Copyright (c) 2019 Manuel Goester, Michael Witt, Klaus Kammerer
Institute of Databases and Information Systems, Ulm University, Germany

Permission is hereby granted, free of charge, to any person obtaining a copy 
of this software and associated documentation files (the "Software"), to deal 
in the Software without restriction, including without limitation the rights 
to use, copy, modify, merge, publish, distribute, sublicense, and/or sell 
copies of the Software, and to permit persons to whom the Software is 
furnished to do so, subject to the following conditions:

The above copyright notice and this permission notice shall be included in 
all copies or substantial portions of the Software.

THE SOFTWARE IS PROVIDED "AS IS", WITHOUT WARRANTY OF ANY KIND, EXPRESS OR 
IMPLIED, INCLUDING BUT NOT LIMITED TO THE WARRANTIES OF MERCHANTABILITY, 
FITNESS FOR A PARTICULAR PURPOSE AND NONINFRINGEMENT. IN NO EVENT SHALL THE 
AUTHORS OR COPYRIGHT HOLDERS BE LIABLE FOR ANY CLAIM, DAMAGES OR OTHER 
LIABILITY, WHETHER IN AN ACTION OF CONTRACT, TORT OR OTHERWISE, ARISING FROM, 
OUT OF OR IN CONNECTION WITH THE SOFTWARE OR THE USE OR OTHER DEALINGS 
IN THE SOFTWARE.
*)
FUNCTION_BLOCK HR_TAKE_W_FROM_CONVEYOR
VAR_INPUT
	w: Workpiece;
END_VAR
VAR_OUTPUT
END_VAR
VAR
	step: INT := 1;
	hr_move: HR_MOVE;
	fin: BOOL := FALSE;
	stepFin: BOOL := FALSE;
END_VAR

fin := FALSE;
CASE step OF
	1:	// forward if not already there
		IF NOT(HR.sCFront) THEN
			HR.mCForward := TRUE;
		ELSE
			HR.mCForward := FALSE;
			step := step + 1;
		END_IF
	2:	// backwards
		IF HR.lbIn THEN
			HR.mCbBackward := TRUE;
		ELSE
			HR.mCbBackward := FALSE;
			step := step + 1; 
		END_IF
	3:	// up
		hr_move(x := 0, y := -26);
		stepFin := hr_move.fin;
		IF stepFin THEN
			step := step + 1;
			stepFin := FALSE;
		END_IF
	4:	// back
		IF NOT(HR.sCBack) THEN
			HR.mCBackward := TRUE;
		ELSE
			HR.mCBackward := FALSE;
			step := step + 1;
		END_IF
	5:	// finished
		fin := TRUE;
		step := 1;
		stepFin := FALSE;
END_CASE

END_FUNCTION_BLOCK

// Device/Application/HR/FBs/HR_PUT_W
(*
	HR puts down a workpiece into rack or at conveyor
	
Copyright (c) 2019 Manuel Goester, Michael Witt, Klaus Kammerer
Institute of Databases and Information Systems, Ulm University, Germany

Permission is hereby granted, free of charge, to any person obtaining a copy 
of this software and associated documentation files (the "Software"), to deal 
in the Software without restriction, including without limitation the rights 
to use, copy, modify, merge, publish, distribute, sublicense, and/or sell 
copies of the Software, and to permit persons to whom the Software is 
furnished to do so, subject to the following conditions:

The above copyright notice and this permission notice shall be included in 
all copies or substantial portions of the Software.

THE SOFTWARE IS PROVIDED "AS IS", WITHOUT WARRANTY OF ANY KIND, EXPRESS OR 
IMPLIED, INCLUDING BUT NOT LIMITED TO THE WARRANTIES OF MERCHANTABILITY, 
FITNESS FOR A PARTICULAR PURPOSE AND NONINFRINGEMENT. IN NO EVENT SHALL THE 
AUTHORS OR COPYRIGHT HOLDERS BE LIABLE FOR ANY CLAIM, DAMAGES OR OTHER 
LIABILITY, WHETHER IN AN ACTION OF CONTRACT, TORT OR OTHERWISE, ARISING FROM, 
OUT OF OR IN CONNECTION WITH THE SOFTWARE OR THE USE OR OTHER DEALINGS 
IN THE SOFTWARE.
*)
FUNCTION_BLOCK HR_PUT_W
VAR_INPUT
END_VAR
VAR_OUTPUT
END_VAR
VAR
	step: INT := 1;
	hr_move: HR_MOVE;
	fin: BOOL := FALSE;
	stepFin: BOOL := FALSE;
END_VAR

CASE step OF
	1:	// forward
		fin := FALSE;
		IF NOT(HR.sCFront) THEN
			HR.mCForward := TRUE;
		ELSE
			HR.mCForward := FALSE;
			step := step + 1;
		END_IF
	2:	// down
		hr_move(x := 0 , y := 16);
		stepFin := hr_move.fin;
		IF stepFin THEN
			step := step + 1;
			stepFin := FALSE;
		END_IF
	3:	// back
		IF NOT(HR.sCBack) THEN
			HR.mCBackward := TRUE;
		ELSE
			HR.mCBackward := FALSE;
			step := step + 1;
		END_IF
	4:	// finished
		fin := TRUE;
		step := 1;
END_CASE

END_FUNCTION_BLOCK

// Device/Application/HR/HR_MULTI_MODE
PROGRAM HR_MULTI_MODE
VAR
	fin: BOOL;
	hr_get: HR_GET_W;
	hr_store: HR_STORE_W;
	hr_put_w_on_conveyor: HR_PUT_W_ON_CONVEYOR;
	
	// for GET_W
	// calibrate y axis of rack every 3th workpiece
	calibrateYAxis: INT := 0;
	calibarteYAxisCounted: BOOL := FALSE;
	step: INT := 1;
	timer: TON;
END_VAR

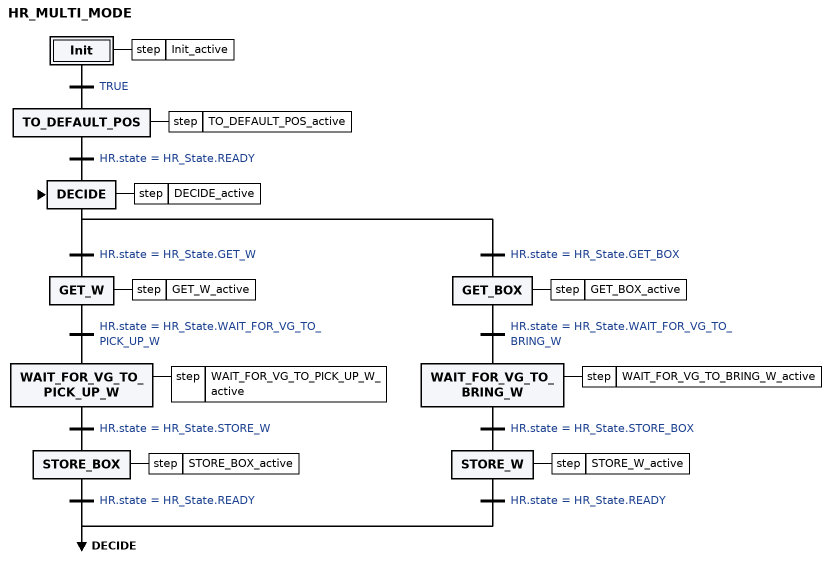
INITIAL_STEP Init:
    Init_active(N);  // step action
END_STEP
TRANSITION FROM Init TO TO_DEFAULT_POS
    := TRUE;
END_TRANSITION
STEP TO_DEFAULT_POS:
    TO_DEFAULT_POS_active(N);  // step action
END_STEP
TRANSITION FROM TO_DEFAULT_POS TO DECIDE
    := HR.state = HR_State.READY;
END_TRANSITION
STEP DECIDE:
    DECIDE_active(N);  // step action
END_STEP
TRANSITION FROM DECIDE TO GET_W
    := HR.state = HR_State.GET_W;
END_TRANSITION
STEP GET_W:
    GET_W_active(N);  // step action
END_STEP
TRANSITION FROM GET_W TO WAIT_FOR_VG_TO_PICK_UP_W
    := HR.state = HR_State.WAIT_FOR_VG_TO_PICK_UP_W;
END_TRANSITION
STEP WAIT_FOR_VG_TO_PICK_UP_W:
    WAIT_FOR_VG_TO_PICK_UP_W_active(N);  // step action
END_STEP
TRANSITION FROM WAIT_FOR_VG_TO_PICK_UP_W TO STORE_BOX
    := HR.state = HR_State.STORE_W;
END_TRANSITION
STEP STORE_BOX:
    STORE_BOX_active(N);  // step action
END_STEP
TRANSITION FROM STORE_BOX TO DECIDE
    := HR.state = HR_State.READY;
END_TRANSITION
TRANSITION FROM DECIDE TO GET_BOX
    := HR.state = HR_State.GET_BOX;
END_TRANSITION
STEP GET_BOX:
    GET_BOX_active(N);  // step action
END_STEP
TRANSITION FROM GET_BOX TO WAIT_FOR_VG_TO_BRING_W
    := HR.state = HR_State.WAIT_FOR_VG_TO_BRING_W;
END_TRANSITION
STEP WAIT_FOR_VG_TO_BRING_W:
    WAIT_FOR_VG_TO_BRING_W_active(N);  // step action
END_STEP
TRANSITION FROM WAIT_FOR_VG_TO_BRING_W TO STORE_W
    := HR.state = HR_State.STORE_BOX;
END_TRANSITION
STEP STORE_W:
    STORE_W_active(N);  // step action
END_STEP
TRANSITION FROM STORE_W TO DECIDE
    := HR.state = HR_State.READY;
END_TRANSITION

ACTION STORE_BOX_active:
(*
Copyright (c) 2019 Manuel Goester, Michael Witt, Klaus Kammerer
Institute of Databases and Information Systems, Ulm University, Germany

Permission is hereby granted, free of charge, to any person obtaining a copy 
of this software and associated documentation files (the "Software"), to deal 
in the Software without restriction, including without limitation the rights 
to use, copy, modify, merge, publish, distribute, sublicense, and/or sell 
copies of the Software, and to permit persons to whom the Software is 
furnished to do so, subject to the following conditions:

The above copyright notice and this permission notice shall be included in 
all copies or substantial portions of the Software.

THE SOFTWARE IS PROVIDED "AS IS", WITHOUT WARRANTY OF ANY KIND, EXPRESS OR 
IMPLIED, INCLUDING BUT NOT LIMITED TO THE WARRANTIES OF MERCHANTABILITY, 
FITNESS FOR A PARTICULAR PURPOSE AND NONINFRINGEMENT. IN NO EVENT SHALL THE 
AUTHORS OR COPYRIGHT HOLDERS BE LIABLE FOR ANY CLAIM, DAMAGES OR OTHER 
LIABILITY, WHETHER IN AN ACTION OF CONTRACT, TORT OR OTHERWISE, ARISING FROM, 
OUT OF OR IN CONNECTION WITH THE SOFTWARE OR THE USE OR OTHER DEALINGS 
IN THE SOFTWARE.
*)
IF NOT fin THEN
	// store box in rack
	hr_store(w := HR.currW);
	fin := hr_store.fin;
ELSE
	fin := FALSE;
	HR.state := HR_State.READY;
END_IF
END_ACTION

ACTION GET_W_active:
(*
Copyright (c) 2019 Manuel Goester, Michael Witt, Klaus Kammerer
Institute of Databases and Information Systems, Ulm University, Germany

Permission is hereby granted, free of charge, to any person obtaining a copy 
of this software and associated documentation files (the "Software"), to deal 
in the Software without restriction, including without limitation the rights 
to use, copy, modify, merge, publish, distribute, sublicense, and/or sell 
copies of the Software, and to permit persons to whom the Software is 
furnished to do so, subject to the following conditions:

The above copyright notice and this permission notice shall be included in 
all copies or substantial portions of the Software.

THE SOFTWARE IS PROVIDED "AS IS", WITHOUT WARRANTY OF ANY KIND, EXPRESS OR 
IMPLIED, INCLUDING BUT NOT LIMITED TO THE WARRANTIES OF MERCHANTABILITY, 
FITNESS FOR A PARTICULAR PURPOSE AND NONINFRINGEMENT. IN NO EVENT SHALL THE 
AUTHORS OR COPYRIGHT HOLDERS BE LIABLE FOR ANY CLAIM, DAMAGES OR OTHER 
LIABILITY, WHETHER IN AN ACTION OF CONTRACT, TORT OR OTHERWISE, ARISING FROM, 
OUT OF OR IN CONNECTION WITH THE SOFTWARE OR THE USE OR OTHER DEALINGS 
IN THE SOFTWARE.
*)
// increment y calibration counter
IF NOT(calibarteYAxisCounted) THEN
	calibrateYAxis := calibrateYAxis + 1;
	calibarteYAxisCounted := TRUE;
END_IF

IF calibrateYAxis >= 3 THEN
	// calibrate y axis
	IF NOT(HR.sVertical) THEN
		HR.mVerticalUp := TRUE;
	ELSE
		Hr.mVerticalUp := FALSE;
		Hr.cY := 0;
		calibrateYAxis := 0;
	END_IF
ELSE
	CASE step OF
		1:
			// get w from rack
			IF NOT fin THEN
				hr_get(w:= HR.currW);
				fin := hr_get.fin;
			ELSE
				fin := FALSE;
				step := step + 1;
			END_IF
		2:
			// put w on conveyor
			hr_put_w_on_conveyor(w := HR.currW);
			fin := hr_put_w_on_conveyor.fin;	
			IF fin THEN
				step := step + 1;
				fin := FALSE;
			END_IF
		3:
			// bring it to VG in conveyor
			IF HR.lbOut THEN
				HR.mCbForward := TRUE;
			ELSE
				// start 1 sec timer to drive conveyor 1 sec longer to be sure that box is at outside pos
				timer(IN:= TRUE, PT := T#1S);
				IF NOT(timer.Q = FALSE AND timer.IN) THEN
					timer(IN:= FALSE);
					HR.mCbForward := FALSE;
					step := step + 1; 
				END_IF
			END_IF
		4:
			// finished
			step := 1;
			HR.state := HR_State.WAIT_FOR_VG_TO_PICK_UP_W;
			calibarteYAxisCounted := FALSE;
			// bend VG pointers to current workpiece of HR
			VG.bIdx := TC.currBatchJobIdx;
			VG.wIdx := TC.batchJobQueue.batchJobs[TC.currBatchJobIdx].nextNotProcessedIdx;
			VG.currW := TC.batchJobQueue.batchJobs[VG.bIdx].workpieces[VG.wIdx];
	END_CASE
END_IF
END_ACTION

ACTION WAIT_FOR_VG_TO_PICK_UP_W_active:
(*
Copyright (c) 2019 Manuel Goester, Michael Witt, Klaus Kammerer
Institute of Databases and Information Systems, Ulm University, Germany

Permission is hereby granted, free of charge, to any person obtaining a copy 
of this software and associated documentation files (the "Software"), to deal 
in the Software without restriction, including without limitation the rights 
to use, copy, modify, merge, publish, distribute, sublicense, and/or sell 
copies of the Software, and to permit persons to whom the Software is 
furnished to do so, subject to the following conditions:

The above copyright notice and this permission notice shall be included in 
all copies or substantial portions of the Software.

THE SOFTWARE IS PROVIDED "AS IS", WITHOUT WARRANTY OF ANY KIND, EXPRESS OR 
IMPLIED, INCLUDING BUT NOT LIMITED TO THE WARRANTIES OF MERCHANTABILITY, 
FITNESS FOR A PARTICULAR PURPOSE AND NONINFRINGEMENT. IN NO EVENT SHALL THE 
AUTHORS OR COPYRIGHT HOLDERS BE LIABLE FOR ANY CLAIM, DAMAGES OR OTHER 
LIABILITY, WHETHER IN AN ACTION OF CONTRACT, TORT OR OTHERWISE, ARISING FROM, 
OUT OF OR IN CONNECTION WITH THE SOFTWARE OR THE USE OR OTHER DEALINGS 
IN THE SOFTWARE.
*)
IF VG.state = VG_State.TO_FUR_PUT_W OR VG.state = VG_State.TO_EJECT THEN
	HR.state := HR_State.STORE_W;
	HR.decidedToTakeANewW := FALSE;
END_IF
END_ACTION

ACTION GET_BOX_active:
(*
Copyright (c) 2019 Manuel Goester, Michael Witt, Klaus Kammerer
Institute of Databases and Information Systems, Ulm University, Germany

Permission is hereby granted, free of charge, to any person obtaining a copy 
of this software and associated documentation files (the "Software"), to deal 
in the Software without restriction, including without limitation the rights 
to use, copy, modify, merge, publish, distribute, sublicense, and/or sell 
copies of the Software, and to permit persons to whom the Software is 
furnished to do so, subject to the following conditions:

The above copyright notice and this permission notice shall be included in 
all copies or substantial portions of the Software.

THE SOFTWARE IS PROVIDED "AS IS", WITHOUT WARRANTY OF ANY KIND, EXPRESS OR 
IMPLIED, INCLUDING BUT NOT LIMITED TO THE WARRANTIES OF MERCHANTABILITY, 
FITNESS FOR A PARTICULAR PURPOSE AND NONINFRINGEMENT. IN NO EVENT SHALL THE 
AUTHORS OR COPYRIGHT HOLDERS BE LIABLE FOR ANY CLAIM, DAMAGES OR OTHER 
LIABILITY, WHETHER IN AN ACTION OF CONTRACT, TORT OR OTHERWISE, ARISING FROM, 
OUT OF OR IN CONNECTION WITH THE SOFTWARE OR THE USE OR OTHER DEALINGS 
IN THE SOFTWARE.
*)
CASE step OF
	1:
		IF NOT fin THEN
			hr_get(w:= HR.currW);
			fin := hr_get.fin;
		ELSE
			step := step + 1;
			fin := FALSE;
		END_IF
	2:
		// put w on conveyor
		hr_put_w_on_conveyor(w := HR.currW);
		fin := hr_put_w_on_conveyor.fin;	
		IF fin THEN
			step := step + 1;
			fin := FALSE;
		END_IF
	3:
		// bring it to VG in conveyor
		IF HR.lbOut THEN
			HR.mCbForward := TRUE;
		ELSE
			// start 1 sec timer to drive conveyor 1 sec longer to be sure that box is at outside pos
			timer(IN:= TRUE, PT := T#1S);
			IF NOT(timer.Q = FALSE AND timer.IN) THEN
				timer(IN:= FALSE);
				HR.mCbForward := FALSE;
				step := step + 1; 
			END_IF
		END_IF
	4:
		// finished
		step := 1;
		HR.state := HR_State.WAIT_FOR_VG_TO_BRING_W;
END_CASE
END_ACTION

ACTION DECIDE_active:
(*
Copyright (c) 2019 Manuel Goester, Michael Witt, Klaus Kammerer
Institute of Databases and Information Systems, Ulm University, Germany

Permission is hereby granted, free of charge, to any person obtaining a copy 
of this software and associated documentation files (the "Software"), to deal 
in the Software without restriction, including without limitation the rights 
to use, copy, modify, merge, publish, distribute, sublicense, and/or sell 
copies of the Software, and to permit persons to whom the Software is 
furnished to do so, subject to the following conditions:

The above copyright notice and this permission notice shall be included in 
all copies or substantial portions of the Software.

THE SOFTWARE IS PROVIDED "AS IS", WITHOUT WARRANTY OF ANY KIND, EXPRESS OR 
IMPLIED, INCLUDING BUT NOT LIMITED TO THE WARRANTIES OF MERCHANTABILITY, 
FITNESS FOR A PARTICULAR PURPOSE AND NONINFRINGEMENT. IN NO EVENT SHALL THE 
AUTHORS OR COPYRIGHT HOLDERS BE LIABLE FOR ANY CLAIM, DAMAGES OR OTHER 
LIABILITY, WHETHER IN AN ACTION OF CONTRACT, TORT OR OTHERWISE, ARISING FROM, 
OUT OF OR IN CONNECTION WITH THE SOFTWARE OR THE USE OR OTHER DEALINGS 
IN THE SOFTWARE.
*)

// if sl positions free or if not free if workpiece will not be ejected 
// AND VG is not storing
// AND HR does not already decided to take a new workpiece
// THEN 
IF ((SL.lbRed AND SL.lbWhite AND SL.lbBlue) OR (SL.currW.format.ejectEnabled AND NOT(SL.currW.state = W_State.NULL))) AND NOT(VG.storeW) AND NOT(decidedToTakeANewW) THEN
	HR.bIdx := 0;
	HR.wIdx := 0;
	HR.currW := TC.nullW;
	HR.decidedToTakeANewW := TRUE;
	VG.storeW := FALSE;
ELSIF HR.decidedToTakeANewW THEN
	// get new w out of rack
	IF TC.state = TC_state.W_LOADED THEN
		// set pointers to make sure that they are set
		Hr.bIdx := TC.currBatchJobIdx;
		Hr.wIdx := TC.batchJobQueue.batchJobs[TC.currBatchJobIdx].nextNotProcessedIdx;
		HR.currW := TC.batchJobQueue.batchJobs[Hr.bIdx].workpieces[Hr.wIdx];
		// workpiece is loaded, start production
		HR.state := HR_State.GET_W;
		// signalise that production starts
		TC.state := TC_State.WAIT_UNTIL_W_FINISHED;
	ELSE
		// no workpiece loaded, load it now
		TC.state := TC_State.LOAD_NEXT_W;
	END_IF
ELSE
	// prevent misconduct when a workpiece is still lying in one of the three spots at SL, although the application got reset
	IF NOT(VG.bIdx = 0) THEN
		// get empty box out of rack
		// set workpiece to get the right box from rack
		IF NOT(SL.lbWhite) OR NOT(SL.lbRed) OR NOT(SL.lbBlue) THEN
			HR.bIdx := SL.bIdx;
			HR.wIdx := SL.wIdx;
			HR.currW := SL.currW;
		ELSE
			HR.bIdx := VG.bIdx;
			HR.wIdx := VG.wIdx;
			HR.currW := VG.currW;
		END_IF
		HR.state := HR_State.GET_BOX;
		// reset flag
		VG.storeW := FALSE;
		END_IF
END_IF
END_ACTION

ACTION STORE_W_active:
(*
Copyright (c) 2019 Manuel Goester, Michael Witt, Klaus Kammerer
Institute of Databases and Information Systems, Ulm University, Germany

Permission is hereby granted, free of charge, to any person obtaining a copy 
of this software and associated documentation files (the "Software"), to deal 
in the Software without restriction, including without limitation the rights 
to use, copy, modify, merge, publish, distribute, sublicense, and/or sell 
copies of the Software, and to permit persons to whom the Software is 
furnished to do so, subject to the following conditions:

The above copyright notice and this permission notice shall be included in 
all copies or substantial portions of the Software.

THE SOFTWARE IS PROVIDED "AS IS", WITHOUT WARRANTY OF ANY KIND, EXPRESS OR 
IMPLIED, INCLUDING BUT NOT LIMITED TO THE WARRANTIES OF MERCHANTABILITY, 
FITNESS FOR A PARTICULAR PURPOSE AND NONINFRINGEMENT. IN NO EVENT SHALL THE 
AUTHORS OR COPYRIGHT HOLDERS BE LIABLE FOR ANY CLAIM, DAMAGES OR OTHER 
LIABILITY, WHETHER IN AN ACTION OF CONTRACT, TORT OR OTHERWISE, ARISING FROM, 
OUT OF OR IN CONNECTION WITH THE SOFTWARE OR THE USE OR OTHER DEALINGS 
IN THE SOFTWARE.
*)
IF NOT fin THEN
	// store workpiece in rack
	hr_store(w := HR.currW);
	fin := hr_store.fin;
ELSE
	fin := FALSE;
	HR.state := HR_State.READY;
END_IF
END_ACTION

ACTION WAIT_FOR_VG_TO_BRING_W_active:
(*
Copyright (c) 2019 Manuel Goester, Michael Witt, Klaus Kammerer
Institute of Databases and Information Systems, Ulm University, Germany

Permission is hereby granted, free of charge, to any person obtaining a copy 
of this software and associated documentation files (the "Software"), to deal 
in the Software without restriction, including without limitation the rights 
to use, copy, modify, merge, publish, distribute, sublicense, and/or sell 
copies of the Software, and to permit persons to whom the Software is 
furnished to do so, subject to the following conditions:

The above copyright notice and this permission notice shall be included in 
all copies or substantial portions of the Software.

THE SOFTWARE IS PROVIDED "AS IS", WITHOUT WARRANTY OF ANY KIND, EXPRESS OR 
IMPLIED, INCLUDING BUT NOT LIMITED TO THE WARRANTIES OF MERCHANTABILITY, 
FITNESS FOR A PARTICULAR PURPOSE AND NONINFRINGEMENT. IN NO EVENT SHALL THE 
AUTHORS OR COPYRIGHT HOLDERS BE LIABLE FOR ANY CLAIM, DAMAGES OR OTHER 
LIABILITY, WHETHER IN AN ACTION OF CONTRACT, TORT OR OTHERWISE, ARISING FROM, 
OUT OF OR IN CONNECTION WITH THE SOFTWARE OR THE USE OR OTHER DEALINGS 
IN THE SOFTWARE.
*)
IF VG.state = VG_State.TO_HR_PUT_W_FINISHED OR HR.currW.format.ejectEnabled THEN
	HR.state := HR_State.STORE_BOX;
END_IF
END_ACTION

ACTION Init_active:
(*
Copyright (c) 2019 Manuel Goester, Michael Witt, Klaus Kammerer
Institute of Databases and Information Systems, Ulm University, Germany

Permission is hereby granted, free of charge, to any person obtaining a copy 
of this software and associated documentation files (the "Software"), to deal 
in the Software without restriction, including without limitation the rights 
to use, copy, modify, merge, publish, distribute, sublicense, and/or sell 
copies of the Software, and to permit persons to whom the Software is 
furnished to do so, subject to the following conditions:

The above copyright notice and this permission notice shall be included in 
all copies or substantial portions of the Software.

THE SOFTWARE IS PROVIDED "AS IS", WITHOUT WARRANTY OF ANY KIND, EXPRESS OR 
IMPLIED, INCLUDING BUT NOT LIMITED TO THE WARRANTIES OF MERCHANTABILITY, 
FITNESS FOR A PARTICULAR PURPOSE AND NONINFRINGEMENT. IN NO EVENT SHALL THE 
AUTHORS OR COPYRIGHT HOLDERS BE LIABLE FOR ANY CLAIM, DAMAGES OR OTHER 
LIABILITY, WHETHER IN AN ACTION OF CONTRACT, TORT OR OTHERWISE, ARISING FROM, 
OUT OF OR IN CONNECTION WITH THE SOFTWARE OR THE USE OR OTHER DEALINGS 
IN THE SOFTWARE.
*)
calibrateYAxis := 0;
calibarteYAxisCounted := FALSE;
END_ACTION

ACTION TO_DEFAULT_POS_active:
(*
Copyright (c) 2019 Manuel Goester, Michael Witt, Klaus Kammerer
Institute of Databases and Information Systems, Ulm University, Germany

Permission is hereby granted, free of charge, to any person obtaining a copy 
of this software and associated documentation files (the "Software"), to deal 
in the Software without restriction, including without limitation the rights 
to use, copy, modify, merge, publish, distribute, sublicense, and/or sell 
copies of the Software, and to permit persons to whom the Software is 
furnished to do so, subject to the following conditions:

The above copyright notice and this permission notice shall be included in 
all copies or substantial portions of the Software.

THE SOFTWARE IS PROVIDED "AS IS", WITHOUT WARRANTY OF ANY KIND, EXPRESS OR 
IMPLIED, INCLUDING BUT NOT LIMITED TO THE WARRANTIES OF MERCHANTABILITY, 
FITNESS FOR A PARTICULAR PURPOSE AND NONINFRINGEMENT. IN NO EVENT SHALL THE 
AUTHORS OR COPYRIGHT HOLDERS BE LIABLE FOR ANY CLAIM, DAMAGES OR OTHER 
LIABILITY, WHETHER IN AN ACTION OF CONTRACT, TORT OR OTHERWISE, ARISING FROM, 
OUT OF OR IN CONNECTION WITH THE SOFTWARE OR THE USE OR OTHER DEALINGS 
IN THE SOFTWARE.
*)
// returns High Rack TOWER to its default start position
// set "ausleger" arm to default position
IF HR.sCBack = FALSE THEN
	HR.mCBackward := TRUE;
ELSE 
	HR.mCBackward := FALSE;
	// set tower vertical position to max UP as well as horizontal position max RIGHT
	IF HR.sHorizontal = FALSE THEN
		HR.mHorizontalRight := TRUE;
	ELSE
		HR.mHorizontalRight := FALSE;
	END_IF
	
	IF HR.sVertical = FALSE THEN
		HR.mVerticalUp := TRUE;
	ELSE
		HR.mVerticalUp := FALSE;
	END_IF
END_IF

IF HR.sHorizontal AND HR.sVertical AND HR.sCBack THEN
	HR.cX := 0;
	HR.cY := 0;
	HR.state := HR_State.READY;
END_IF
END_ACTION

END_PROGRAM

// Device/Application/HR/HR_SORTING_MODE
PROGRAM HR_SORTING_MODE
VAR
	hr_switch_ws: HR_SWITCH_WS;
	fin: BOOL;
END_VAR

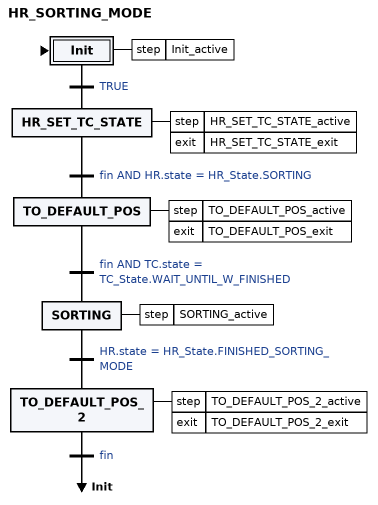
INITIAL_STEP Init:
    Init_active(N);  // step action
END_STEP
TRANSITION FROM Init TO HR_SET_TC_STATE
    := TRUE;
END_TRANSITION
STEP HR_SET_TC_STATE:
    HR_SET_TC_STATE_active(N);  // step action
    HR_SET_TC_STATE_exit(P0);  // exit action
END_STEP
TRANSITION FROM HR_SET_TC_STATE TO TO_DEFAULT_POS
    := fin AND HR.state = HR_State.SORTING;
END_TRANSITION
STEP TO_DEFAULT_POS:
    TO_DEFAULT_POS_active(N);  // step action
    TO_DEFAULT_POS_exit(P0);  // exit action
END_STEP
TRANSITION FROM TO_DEFAULT_POS TO SORTING
    := fin AND TC.state = TC_State.WAIT_UNTIL_W_FINISHED;
END_TRANSITION
STEP SORTING:
    SORTING_active(N);  // step action
END_STEP
TRANSITION FROM SORTING TO TO_DEFAULT_POS_2
    := HR.state = HR_State.FINISHED_SORTING_MODE;
END_TRANSITION
STEP TO_DEFAULT_POS_2:
    TO_DEFAULT_POS_2_active(N);  // step action
    TO_DEFAULT_POS_2_exit(P0);  // exit action
END_STEP
TRANSITION FROM TO_DEFAULT_POS_2 TO Init
    := fin;
END_TRANSITION

ACTION SORTING_active:
(*
Copyright (c) 2019 Manuel Goester, Michael Witt, Klaus Kammerer
Institute of Databases and Information Systems, Ulm University, Germany

Permission is hereby granted, free of charge, to any person obtaining a copy 
of this software and associated documentation files (the "Software"), to deal 
in the Software without restriction, including without limitation the rights 
to use, copy, modify, merge, publish, distribute, sublicense, and/or sell 
copies of the Software, and to permit persons to whom the Software is 
furnished to do so, subject to the following conditions:

The above copyright notice and this permission notice shall be included in 
all copies or substantial portions of the Software.

THE SOFTWARE IS PROVIDED "AS IS", WITHOUT WARRANTY OF ANY KIND, EXPRESS OR 
IMPLIED, INCLUDING BUT NOT LIMITED TO THE WARRANTIES OF MERCHANTABILITY, 
FITNESS FOR A PARTICULAR PURPOSE AND NONINFRINGEMENT. IN NO EVENT SHALL THE 
AUTHORS OR COPYRIGHT HOLDERS BE LIABLE FOR ANY CLAIM, DAMAGES OR OTHER 
LIABILITY, WHETHER IN AN ACTION OF CONTRACT, TORT OR OTHERWISE, ARISING FROM, 
OUT OF OR IN CONNECTION WITH THE SOFTWARE OR THE USE OR OTHER DEALINGS 
IN THE SOFTWARE.
*)
IF NOT(fin) THEN
	hr_switch_ws(w1 := TC.batchJobQueue.batchJobs[TC.currBatchJobIdx].workpieces[TC.batchJobQueue.batchJobs[TC.currBatchJobIdx].nextNotProcessedIdx], w2 := TC.batchJobQueue.batchJobs[TC.currBatchJobIdx].workpieces[TC.batchJobQueue.batchJobs[TC.currBatchJobIdx].nextNotProcessedIdx+1]);
	fin := hr_switch_ws.fin;
ELSE
	// sorting finished
	fin := FALSE;
	HR.state := HR_State.FINISHED_SORTING_MODE;
END_IF
END_ACTION

ACTION TO_DEFAULT_POS_exit:
(*
Copyright (c) 2019 Manuel Goester, Michael Witt, Klaus Kammerer
Institute of Databases and Information Systems, Ulm University, Germany

Permission is hereby granted, free of charge, to any person obtaining a copy 
of this software and associated documentation files (the "Software"), to deal 
in the Software without restriction, including without limitation the rights 
to use, copy, modify, merge, publish, distribute, sublicense, and/or sell 
copies of the Software, and to permit persons to whom the Software is 
furnished to do so, subject to the following conditions:

The above copyright notice and this permission notice shall be included in 
all copies or substantial portions of the Software.

THE SOFTWARE IS PROVIDED "AS IS", WITHOUT WARRANTY OF ANY KIND, EXPRESS OR 
IMPLIED, INCLUDING BUT NOT LIMITED TO THE WARRANTIES OF MERCHANTABILITY, 
FITNESS FOR A PARTICULAR PURPOSE AND NONINFRINGEMENT. IN NO EVENT SHALL THE 
AUTHORS OR COPYRIGHT HOLDERS BE LIABLE FOR ANY CLAIM, DAMAGES OR OTHER 
LIABILITY, WHETHER IN AN ACTION OF CONTRACT, TORT OR OTHERWISE, ARISING FROM, 
OUT OF OR IN CONNECTION WITH THE SOFTWARE OR THE USE OR OTHER DEALINGS 
IN THE SOFTWARE.
*)
fin := FALSE;
END_ACTION

ACTION TO_DEFAULT_POS_active:
(*
Copyright (c) 2019 Manuel Goester, Michael Witt, Klaus Kammerer
Institute of Databases and Information Systems, Ulm University, Germany

Permission is hereby granted, free of charge, to any person obtaining a copy 
of this software and associated documentation files (the "Software"), to deal 
in the Software without restriction, including without limitation the rights 
to use, copy, modify, merge, publish, distribute, sublicense, and/or sell 
copies of the Software, and to permit persons to whom the Software is 
furnished to do so, subject to the following conditions:

The above copyright notice and this permission notice shall be included in 
all copies or substantial portions of the Software.

THE SOFTWARE IS PROVIDED "AS IS", WITHOUT WARRANTY OF ANY KIND, EXPRESS OR 
IMPLIED, INCLUDING BUT NOT LIMITED TO THE WARRANTIES OF MERCHANTABILITY, 
FITNESS FOR A PARTICULAR PURPOSE AND NONINFRINGEMENT. IN NO EVENT SHALL THE 
AUTHORS OR COPYRIGHT HOLDERS BE LIABLE FOR ANY CLAIM, DAMAGES OR OTHER 
LIABILITY, WHETHER IN AN ACTION OF CONTRACT, TORT OR OTHERWISE, ARISING FROM, 
OUT OF OR IN CONNECTION WITH THE SOFTWARE OR THE USE OR OTHER DEALINGS 
IN THE SOFTWARE.
*)
// get HR to its default position
IF HR.sCBack = FALSE THEN
	HR.mCBackward := TRUE;
ELSE 
	HR.mCBackward := FALSE;
	// set tower vertical position to max UP as well as horizontal position max RIGHT
	IF HR.sHorizontal = FALSE THEN
		HR.mHorizontalRight := TRUE;
	ELSE
		HR.mHorizontalRight := FALSE;
		HR.cX := 0;
	END_IF
	
	IF HR.sVertical = FALSE THEN
		HR.mVerticalUp := TRUE;
	ELSE
		HR.mVerticalUp := FALSE;
		HR.cY := 0;
	END_IF
END_IF

IF HR.sHorizontal AND HR.sVertical AND HR.sCBack THEN
	// finished
	fin := TRUE;
END_IF
END_ACTION

ACTION Init_active:

END_ACTION

ACTION HR_SET_TC_STATE_active:
(*
Copyright (c) 2019 Manuel Goester, Michael Witt, Klaus Kammerer
Institute of Databases and Information Systems, Ulm University, Germany

Permission is hereby granted, free of charge, to any person obtaining a copy 
of this software and associated documentation files (the "Software"), to deal 
in the Software without restriction, including without limitation the rights 
to use, copy, modify, merge, publish, distribute, sublicense, and/or sell 
copies of the Software, and to permit persons to whom the Software is 
furnished to do so, subject to the following conditions:

The above copyright notice and this permission notice shall be included in 
all copies or substantial portions of the Software.

THE SOFTWARE IS PROVIDED "AS IS", WITHOUT WARRANTY OF ANY KIND, EXPRESS OR 
IMPLIED, INCLUDING BUT NOT LIMITED TO THE WARRANTIES OF MERCHANTABILITY, 
FITNESS FOR A PARTICULAR PURPOSE AND NONINFRINGEMENT. IN NO EVENT SHALL THE 
AUTHORS OR COPYRIGHT HOLDERS BE LIABLE FOR ANY CLAIM, DAMAGES OR OTHER 
LIABILITY, WHETHER IN AN ACTION OF CONTRACT, TORT OR OTHERWISE, ARISING FROM, 
OUT OF OR IN CONNECTION WITH THE SOFTWARE OR THE USE OR OTHER DEALINGS 
IN THE SOFTWARE.
*)
IF NOT(fin) THEN
	IF TC.state = TC_State.W_LOADED THEN
		TC.state := TC_State.WAIT_UNTIL_W_FINISHED;
		fin := TRUE;
	ELSE
		// load a new workpiece
		TC.state := TC_State.LOAD_NEXT_W;
	END_IF
END_IF
END_ACTION

ACTION HR_SET_TC_STATE_exit:
(*
Copyright (c) 2019 Manuel Goester, Michael Witt, Klaus Kammerer
Institute of Databases and Information Systems, Ulm University, Germany

Permission is hereby granted, free of charge, to any person obtaining a copy 
of this software and associated documentation files (the "Software"), to deal 
in the Software without restriction, including without limitation the rights 
to use, copy, modify, merge, publish, distribute, sublicense, and/or sell 
copies of the Software, and to permit persons to whom the Software is 
furnished to do so, subject to the following conditions:

The above copyright notice and this permission notice shall be included in 
all copies or substantial portions of the Software.

THE SOFTWARE IS PROVIDED "AS IS", WITHOUT WARRANTY OF ANY KIND, EXPRESS OR 
IMPLIED, INCLUDING BUT NOT LIMITED TO THE WARRANTIES OF MERCHANTABILITY, 
FITNESS FOR A PARTICULAR PURPOSE AND NONINFRINGEMENT. IN NO EVENT SHALL THE 
AUTHORS OR COPYRIGHT HOLDERS BE LIABLE FOR ANY CLAIM, DAMAGES OR OTHER 
LIABILITY, WHETHER IN AN ACTION OF CONTRACT, TORT OR OTHERWISE, ARISING FROM, 
OUT OF OR IN CONNECTION WITH THE SOFTWARE OR THE USE OR OTHER DEALINGS 
IN THE SOFTWARE.
*)
fin := FALSE;
END_ACTION

ACTION TO_DEFAULT_POS_2_exit:
(*
Copyright (c) 2019 Manuel Goester, Michael Witt, Klaus Kammerer
Institute of Databases and Information Systems, Ulm University, Germany

Permission is hereby granted, free of charge, to any person obtaining a copy 
of this software and associated documentation files (the "Software"), to deal 
in the Software without restriction, including without limitation the rights 
to use, copy, modify, merge, publish, distribute, sublicense, and/or sell 
copies of the Software, and to permit persons to whom the Software is 
furnished to do so, subject to the following conditions:

The above copyright notice and this permission notice shall be included in 
all copies or substantial portions of the Software.

THE SOFTWARE IS PROVIDED "AS IS", WITHOUT WARRANTY OF ANY KIND, EXPRESS OR 
IMPLIED, INCLUDING BUT NOT LIMITED TO THE WARRANTIES OF MERCHANTABILITY, 
FITNESS FOR A PARTICULAR PURPOSE AND NONINFRINGEMENT. IN NO EVENT SHALL THE 
AUTHORS OR COPYRIGHT HOLDERS BE LIABLE FOR ANY CLAIM, DAMAGES OR OTHER 
LIABILITY, WHETHER IN AN ACTION OF CONTRACT, TORT OR OTHERWISE, ARISING FROM, 
OUT OF OR IN CONNECTION WITH THE SOFTWARE OR THE USE OR OTHER DEALINGS 
IN THE SOFTWARE.
*)
fin := FALSE;
END_ACTION

ACTION TO_DEFAULT_POS_2_active:
(*
Copyright (c) 2019 Manuel Goester, Michael Witt, Klaus Kammerer
Institute of Databases and Information Systems, Ulm University, Germany

Permission is hereby granted, free of charge, to any person obtaining a copy 
of this software and associated documentation files (the "Software"), to deal 
in the Software without restriction, including without limitation the rights 
to use, copy, modify, merge, publish, distribute, sublicense, and/or sell 
copies of the Software, and to permit persons to whom the Software is 
furnished to do so, subject to the following conditions:

The above copyright notice and this permission notice shall be included in 
all copies or substantial portions of the Software.

THE SOFTWARE IS PROVIDED "AS IS", WITHOUT WARRANTY OF ANY KIND, EXPRESS OR 
IMPLIED, INCLUDING BUT NOT LIMITED TO THE WARRANTIES OF MERCHANTABILITY, 
FITNESS FOR A PARTICULAR PURPOSE AND NONINFRINGEMENT. IN NO EVENT SHALL THE 
AUTHORS OR COPYRIGHT HOLDERS BE LIABLE FOR ANY CLAIM, DAMAGES OR OTHER 
LIABILITY, WHETHER IN AN ACTION OF CONTRACT, TORT OR OTHERWISE, ARISING FROM, 
OUT OF OR IN CONNECTION WITH THE SOFTWARE OR THE USE OR OTHER DEALINGS 
IN THE SOFTWARE.
*)
// get HR to its default position
// needed, if a job multi / single mode batch job will be executed after ths batch
IF HR.sCBack = FALSE THEN
	HR.mCBackward := TRUE;
ELSE 
	HR.mCBackward := FALSE;
	// set tower vertical position to max UP as well as horizontal position max RIGHT
	IF HR.sHorizontal = FALSE THEN
		HR.mHorizontalRight := TRUE;
	ELSE
		HR.mHorizontalRight := FALSE;
		HR.cX := 0;
	END_IF
	
	IF HR.sVertical = FALSE THEN
		HR.mVerticalUp := TRUE;
	ELSE
		HR.mVerticalUp := FALSE;
		HR.cY := 0;
	END_IF
END_IF

IF HR.sHorizontal AND HR.sVertical AND HR.sCBack THEN
	// finished
	fin := TRUE;
END_IF
END_ACTION

END_PROGRAM

// Device/Application/HR/FBs/HR_SWITCH_WS
(*
	This Function Block gets two workpieces as input and switches their positions in the rack
	
Copyright (c) 2019 Manuel Goester, Michael Witt, Klaus Kammerer
Institute of Databases and Information Systems, Ulm University, Germany

Permission is hereby granted, free of charge, to any person obtaining a copy 
of this software and associated documentation files (the "Software"), to deal 
in the Software without restriction, including without limitation the rights 
to use, copy, modify, merge, publish, distribute, sublicense, and/or sell 
copies of the Software, and to permit persons to whom the Software is 
furnished to do so, subject to the following conditions:

The above copyright notice and this permission notice shall be included in 
all copies or substantial portions of the Software.

THE SOFTWARE IS PROVIDED "AS IS", WITHOUT WARRANTY OF ANY KIND, EXPRESS OR 
IMPLIED, INCLUDING BUT NOT LIMITED TO THE WARRANTIES OF MERCHANTABILITY, 
FITNESS FOR A PARTICULAR PURPOSE AND NONINFRINGEMENT. IN NO EVENT SHALL THE 
AUTHORS OR COPYRIGHT HOLDERS BE LIABLE FOR ANY CLAIM, DAMAGES OR OTHER 
LIABILITY, WHETHER IN AN ACTION OF CONTRACT, TORT OR OTHERWISE, ARISING FROM, 
OUT OF OR IN CONNECTION WITH THE SOFTWARE OR THE USE OR OTHER DEALINGS 
IN THE SOFTWARE.
*)
FUNCTION_BLOCK HR_SWITCH_WS
VAR_INPUT
	// first workpiece
	w1: Workpiece;
	// second workpiece
	w2: Workpiece;
END_VAR
VAR_OUTPUT
END_VAR
VAR
	stepFin : BOOL;
	step: INT := 1;
	hr_move_to_pos: HR_MOVE_TO_POS;
	hr_get_w: HR_GET_W;
	hr_take_w: HR_TAKE_W;
	hr_put_w: HR_PUT_W;
	fin: BOOL;
END_VAR

fin := FALSE;
CASE step OF
	1:	// get w1 out of rack and bring it to conveyor
		IF NOT(stepFin) THEN
			hr_get_w(w := w1);
			stepFin := hr_get_w.fin;
		ELSE
			stepFin := FALSE;
			step := step + 1;
		END_IF
	2:	// put down w1 at conveyor
		IF NOT(stepFin) THEN
			hr_put_w();
			stepFin := hr_put_w.fin;
		ELSE
			stepFin := FALSE;
			step := step + 1;
		END_IF
	3:	// move to w2 position in rack
		IF NOT(stepFin) THEN
			hr_move_to_pos(pos := w2.startPos, upOrDown := RackPos.DOWN);	
			stepFin := hr_move_to_pos.fin;
		ELSE
			stepFin := FALSE;
			step := step + 1;
		END_IF
	4:	// pick up w2
		IF NOT(stepFin) THEN
			hr_take_w();
			stepFin := hr_take_w.fin;
		ELSE
			stepFin := FALSE;
			step := step + 1;
		END_IF
	5:	// move to w1 start-position in rack
		IF NOT(stepFin) THEN
			hr_move_to_pos(pos := w1.startPos, upOrDown := RackPos.UP);	
			stepFin := hr_move_to_pos.fin;
		ELSE
			stepFin := FALSE;
			step := step + 1;
		END_IF
	6:	// put down w2 in rack
		IF NOT(stepFin) THEN
			hr_put_w();
			stepFin := hr_put_w.fin;
		ELSE
			stepFin := FALSE;
			step := step + 1;
		END_IF
	7:	// move to conveyor
		IF NOT(stepFin) THEN
			hr_move_to_pos(pos := RackPos.CONVEYOR, upOrDown := RackPos.DOWN);	
			stepFin := hr_move_to_pos.fin;
		ELSE
			stepFin := FALSE;
			step := step + 1;
		END_IF
	8:	// pick up w1 at conveyor
		IF NOT(stepFin) THEN
			hr_take_w();
			stepFin := hr_take_w.fin;
		ELSE
			stepFin := FALSE;
			step := step + 1;
		END_IF
	9:	// move to rack to start-position of w2
		IF NOT(stepFin) THEN
			hr_move_to_pos(pos := w2.startPos, upOrDown := RackPos.UP);	
			stepFin := hr_move_to_pos.fin;
		ELSE
			stepFin := FALSE;
			step := step + 1;
		END_IF
	10:	// put down w1 in rack
		IF NOT(stepFin) THEN
			hr_put_w();
			stepFin := hr_put_w.fin;
		ELSE
			stepFin := FALSE;
			step := step + 1;
		END_IF
	11:	// finished
		fin := TRUE;
		step := 1;
END_CASE

END_FUNCTION_BLOCK

// Device/Application/TC/FUNs/addBatchJobToQueue
(*
	Adds a BatchJob to TC.BatchJobQueue
	
Copyright (c) 2019 Manuel Goester, Michael Witt, Klaus Kammerer
Institute of Databases and Information Systems, Ulm University, Germany

Permission is hereby granted, free of charge, to any person obtaining a copy 
of this software and associated documentation files (the "Software"), to deal 
in the Software without restriction, including without limitation the rights 
to use, copy, modify, merge, publish, distribute, sublicense, and/or sell 
copies of the Software, and to permit persons to whom the Software is 
furnished to do so, subject to the following conditions:

The above copyright notice and this permission notice shall be included in 
all copies or substantial portions of the Software.

THE SOFTWARE IS PROVIDED "AS IS", WITHOUT WARRANTY OF ANY KIND, EXPRESS OR 
IMPLIED, INCLUDING BUT NOT LIMITED TO THE WARRANTIES OF MERCHANTABILITY, 
FITNESS FOR A PARTICULAR PURPOSE AND NONINFRINGEMENT. IN NO EVENT SHALL THE 
AUTHORS OR COPYRIGHT HOLDERS BE LIABLE FOR ANY CLAIM, DAMAGES OR OTHER 
LIABILITY, WHETHER IN AN ACTION OF CONTRACT, TORT OR OTHERWISE, ARISING FROM, 
OUT OF OR IN CONNECTION WITH THE SOFTWARE OR THE USE OR OTHER DEALINGS 
IN THE SOFTWARE.
*)
FUNCTION addBatchJobToQueue : BOOL
VAR_INPUT
	// The BatchJob which will be added
	batchJob: BatchJob;
END_VAR
VAR
END_VAR

IF 1 <= TC.batchJobQueue.nextFreePos AND TC.batchJobQueue.nextFreePos <= 20 THEN
	TC.batchJobQueue.batchJobs[TC.batchJobQueue.nextFreePos] := batchJob;
	TC.batchJobQueue.nextFreePos := TC.batchJobQueue.nextFreePos + 1;
	TC.batchJobQueue.amountBatchJobs := TC.batchJobQueue.amountBatchJobs + 1;
	IF TC.batchJobQueue.amountBatchJobs = 20 THEN
		TC.batchJobQueue.full := TRUE;
	ELSE
		TC.batchJobQueue.full := FALSE;
	END_IF
	addBatchJobToQueue := TRUE;
ELSE
	// Batch Job Queue already full
	addBatchJobToQueue := FALSE;	
END_IF
RETURN;

END_FUNCTION

// Device/Application/TC/FUNs/newFormat
(*
	Constructor for Format
	A Format defines the options for a production of a workpiece
	
Copyright (c) 2019 Manuel Goester, Michael Witt, Klaus Kammerer
Institute of Databases and Information Systems, Ulm University, Germany

Permission is hereby granted, free of charge, to any person obtaining a copy 
of this software and associated documentation files (the "Software"), to deal 
in the Software without restriction, including without limitation the rights 
to use, copy, modify, merge, publish, distribute, sublicense, and/or sell 
copies of the Software, and to permit persons to whom the Software is 
furnished to do so, subject to the following conditions:

The above copyright notice and this permission notice shall be included in 
all copies or substantial portions of the Software.

THE SOFTWARE IS PROVIDED "AS IS", WITHOUT WARRANTY OF ANY KIND, EXPRESS OR 
IMPLIED, INCLUDING BUT NOT LIMITED TO THE WARRANTIES OF MERCHANTABILITY, 
FITNESS FOR A PARTICULAR PURPOSE AND NONINFRINGEMENT. IN NO EVENT SHALL THE 
AUTHORS OR COPYRIGHT HOLDERS BE LIABLE FOR ANY CLAIM, DAMAGES OR OTHER 
LIABILITY, WHETHER IN AN ACTION OF CONTRACT, TORT OR OTHERWISE, ARISING FROM, 
OUT OF OR IN CONNECTION WITH THE SOFTWARE OR THE USE OR OTHER DEALINGS 
IN THE SOFTWARE.
*)
FUNCTION newFormat : Format
VAR_INPUT
	furEnabled: BOOL;
	sawEnabled: BOOL;
	colorCheckEnabled: BOOL;
	ejectEnabled: BOOL;
	
	furDuration: TIME;
	sawDuration: TIME;
END_VAR
VAR
END_VAR

newFormat.furEnabled := furEnabled;
newFormat.sawEnabled := sawEnabled;
newFormat.colorCheckEnabled := colorCheckEnabled;
newFormat.ejectEnabled := ejectEnabled;
newFormat.furDuration := furDuration;
newFormat.sawDuration := sawDuration;
RETURN;

END_FUNCTION

// Device/Application/TC/FUNs/newWorkpiece
(*
	Constructor for Workpiece 
	
Copyright (c) 2019 Manuel Goester, Michael Witt, Klaus Kammerer
Institute of Databases and Information Systems, Ulm University, Germany

Permission is hereby granted, free of charge, to any person obtaining a copy 
of this software and associated documentation files (the "Software"), to deal 
in the Software without restriction, including without limitation the rights 
to use, copy, modify, merge, publish, distribute, sublicense, and/or sell 
copies of the Software, and to permit persons to whom the Software is 
furnished to do so, subject to the following conditions:

The above copyright notice and this permission notice shall be included in 
all copies or substantial portions of the Software.

THE SOFTWARE IS PROVIDED "AS IS", WITHOUT WARRANTY OF ANY KIND, EXPRESS OR 
IMPLIED, INCLUDING BUT NOT LIMITED TO THE WARRANTIES OF MERCHANTABILITY, 
FITNESS FOR A PARTICULAR PURPOSE AND NONINFRINGEMENT. IN NO EVENT SHALL THE 
AUTHORS OR COPYRIGHT HOLDERS BE LIABLE FOR ANY CLAIM, DAMAGES OR OTHER 
LIABILITY, WHETHER IN AN ACTION OF CONTRACT, TORT OR OTHERWISE, ARISING FROM, 
OUT OF OR IN CONNECTION WITH THE SOFTWARE OR THE USE OR OTHER DEALINGS 
IN THE SOFTWARE.
*)
FUNCTION newWorkpiece : Workpiece
VAR_INPUT
	// color of the workpiece: red, blue, white or unknown
	color: STRING[7];
	
	// state at start: 1ij, i = vertical pos in rack at begin, j = horizontal pos in rack at begin
	state: W_State;
	
	startPos: RackPos;

	endPos: RackPos;
	
	// format for this workpiece
	format: Format;
END_VAR
VAR
END_VAR

newWorkpiece.color := color;
newWorkpiece.format := format;
newWorkpiece.startPos := startPos;
newWorkpiece.endPos := endPos;
newWorkpiece.sortingLinePos := -1;
newWorkpiece.linePos := 0;
newWorkpiece.state := state;
RETURN;

END_FUNCTION

// Device/Application/TC/FUNs/newBatchJob
(*
	Constructor of a BatchJob
	
Copyright (c) 2019 Manuel Goester, Michael Witt, Klaus Kammerer
Institute of Databases and Information Systems, Ulm University, Germany

Permission is hereby granted, free of charge, to any person obtaining a copy 
of this software and associated documentation files (the "Software"), to deal 
in the Software without restriction, including without limitation the rights 
to use, copy, modify, merge, publish, distribute, sublicense, and/or sell 
copies of the Software, and to permit persons to whom the Software is 
furnished to do so, subject to the following conditions:

The above copyright notice and this permission notice shall be included in 
all copies or substantial portions of the Software.

THE SOFTWARE IS PROVIDED "AS IS", WITHOUT WARRANTY OF ANY KIND, EXPRESS OR 
IMPLIED, INCLUDING BUT NOT LIMITED TO THE WARRANTIES OF MERCHANTABILITY, 
FITNESS FOR A PARTICULAR PURPOSE AND NONINFRINGEMENT. IN NO EVENT SHALL THE 
AUTHORS OR COPYRIGHT HOLDERS BE LIABLE FOR ANY CLAIM, DAMAGES OR OTHER 
LIABILITY, WHETHER IN AN ACTION OF CONTRACT, TORT OR OTHERWISE, ARISING FROM, 
OUT OF OR IN CONNECTION WITH THE SOFTWARE OR THE USE OR OTHER DEALINGS 
IN THE SOFTWARE.
*)
FUNCTION newBatchJob : BatchJob
VAR_INPUT
	// amount of workpieces in batch job
	batchSize: INT;
	
	// workpieces being processed
	workpieces: ARRAY [1..9] OF Workpiece;
	
	// type of execution: single, multi or sorting
	mode: ExecutionMode;
END_VAR
VAR
	placeFound: BOOL := FALSE;
	wsFull: BOOL := FALSE;
	i: INT := 1;
	sysTime: RTC;
END_VAR

newBatchJob.batchSize := batchSize;
newBatchJob.workpieces := workpieces;
newBatchJob.mode := mode;

// Search for next free position in workpieces. If there is no free position, set nextFreeWPos to -1
WHILE NOT(placeFound) AND NOT(wsFull) DO
	IF workpieces[i].state = W_State.NULL THEN
		placeFound := TRUE;
		newBatchJob.nextFreeWPos := i;
	ELSIF i > newBatchJob.batchSize THEN
		wsFull := TRUE;
		newBatchJob.nextFreeWPos := -1;
	ELSE
		i := i + 1;
	END_IF
END_WHILE

newBatchJob.nextNotProcessedIdx := 1;
newBatchJob.amountFinishedW := 0;
newBatchJob.duration := T#0S;
newBatchJob.pauseDuration := T#0S;
newBatchJob.state := BatchJobState.WAITING;
// current system time
newBatchJob.timeCreated := sysTime.CDT;
RETURN;

END_FUNCTION

// Device/Application/TC/FUNs/addWorkpieceToBatchJob
(*
	Adds the workpiece w to the batchJobs queue, if there is a free place in the queue
	
Copyright (c) 2019 Manuel Goester, Michael Witt, Klaus Kammerer
Institute of Databases and Information Systems, Ulm University, Germany

Permission is hereby granted, free of charge, to any person obtaining a copy 
of this software and associated documentation files (the "Software"), to deal 
in the Software without restriction, including without limitation the rights 
to use, copy, modify, merge, publish, distribute, sublicense, and/or sell 
copies of the Software, and to permit persons to whom the Software is 
furnished to do so, subject to the following conditions:

The above copyright notice and this permission notice shall be included in 
all copies or substantial portions of the Software.

THE SOFTWARE IS PROVIDED "AS IS", WITHOUT WARRANTY OF ANY KIND, EXPRESS OR 
IMPLIED, INCLUDING BUT NOT LIMITED TO THE WARRANTIES OF MERCHANTABILITY, 
FITNESS FOR A PARTICULAR PURPOSE AND NONINFRINGEMENT. IN NO EVENT SHALL THE 
AUTHORS OR COPYRIGHT HOLDERS BE LIABLE FOR ANY CLAIM, DAMAGES OR OTHER 
LIABILITY, WHETHER IN AN ACTION OF CONTRACT, TORT OR OTHERWISE, ARISING FROM, 
OUT OF OR IN CONNECTION WITH THE SOFTWARE OR THE USE OR OTHER DEALINGS 
IN THE SOFTWARE.
*)
FUNCTION addWorkpieceToBatchJob : BOOL
VAR_INPUT
	// the batch job
	batchJob: BatchJob;
	
	// the workpiece to be added to the batch jobs queue
	w: workpiece;
END_VAR
VAR
	
END_VAR

IF batchJob.nextFreeWPos >= 1 AND batchJob.nextFreeWPos <= 9 THEN
	// free place available
	batchJob.workpieces[batchJob.nextFreeWPos] := w;
	batchJob.nextFreeWPos := batchJob.nextFreeWPos + 1;
	batchJob.batchSize := batchJob.batchSize + 1;
	AddWorkpieceToBatchJob := TRUE;
ELSE
	// queue full
	AddWorkpieceToBatchJob := FALSE;
END_IF
RETURN;

END_FUNCTION

// Device/Application/Visu
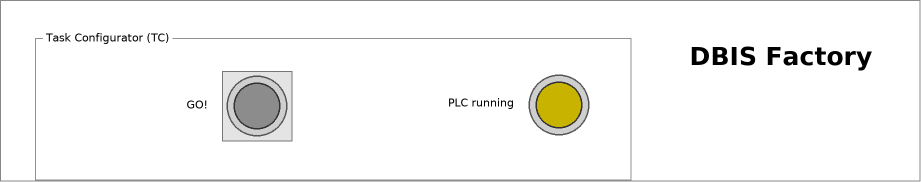
VISUALIZATION Visu  // 921x182
    GroupBox (35,30 596x150), "Task Configurator (TC)"
        Lamp1 (489,40 70x70), variable: is_plc_running, style: Lamp-Lamp1-Yellow
        Label (332,58 150x30), "PLC running"
        PushSwitch (187,41 70x70), variable: TC_POU.started, behaviour: TOGGLE, style: Switch-PushSwitch-Gray
        Label (26,60 150x30), "GO!"
    Label (643,31 276x50), "DBIS Factory"
END_VISUALIZATION
